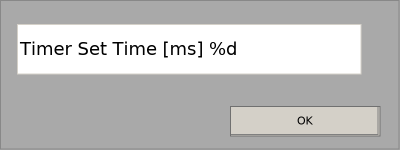
VISUALIZATION DialogTimer_ColdCut  // 400x150
    Button (230,106 150x30), "OK"
        OnMouseClick: CloseDialog Dialog=DialogTimer_ColdCut, Result=OK, NumpadKeypadSet=True
    Textfield (17,24 344x50), "Timer Set Time [ms] %d", text variable: PersistentStruct.TimeColdCutPressDown
        OnMouseClick: write the text variable via Edit
END_VISUALIZATION

(* stored: Version 1.1.0.1, ProductVersion 3.1.4024.3
   Visu DialogTimer_ColdCut: Id {7ec4d096-5ad0-427b-a774-4d917bb3e1f3} *)
